INTERFACE I_GeometryWriter

METHOD AddArc : BOOL
VAR_INPUT
    TargetX    : LREAL;
    TargetY    : LREAL;
    CenterX    : LREAL;
    CenterY    : LREAL;
    Velo       : LREAL;
    Clockwise  : BOOL; 
END_VAR
END_METHOD

METHOD AddLine : BOOL
VAR_INPUT
    TargetX : LREAL;
    TargetY : LREAL;
    Velo    : LREAL;
END_VAR
END_METHOD

METHOD AddStartPoint : BOOL
VAR_INPUT
    TargetX : LREAL;
    TargetY : LREAL;
END_VAR
END_METHOD

METHOD Clear : BOOL
VAR_INPUT
END_VAR
END_METHOD

METHOD EnableTangentialFollowing : BOOL
VAR_INPUT
END_VAR
END_METHOD

METHOD EndTable : BOOL
VAR_INPUT
END_VAR
END_METHOD

END_INTERFACE

(* stored: Version 1.1.0.1, ProductVersion 3.1.4024.15
   Itf I_GeometryWriter: Id {30dc15d7-2c56-44a4-aaea-17b7aa8b5c9b}
   Method AddArc: Id {a72e30e6-e984-4c37-9121-f29f6b1927b6}
   Method AddLine: Id {f4f04758-1e9c-46c2-a655-389290c6ffc8}
   Method AddStartPoint: Id {a9c855e3-b199-4571-b454-c231e9f1c099}
   Method Clear: Id {6886b5bf-f669-42e8-933c-2f73bf76f494}
   Method EnableTangentialFollowing: Id {31f985d8-d88b-4600-b935-ef1d86cff651}
   Method EndTable: Id {5d7b8dfb-7103-409c-b6f4-152577166389} *)
